// This function has been automatically generated from the project information.
{attribute 'signature_flag' := '1073741824'}
{attribute 'TcGenerated'}
{attribute 'no-analysis'}
FUNCTION F_GetTitle : WSTRING
VAR_INPUT
	
END_VAR

F_GetTitle := "Motion Library";

END_FUNCTION

(* stored: Version 1.1.0.1
   POU F_GetTitle: Id {c210cf97-aa66-408b-beb4-809f283b95e5}, SpecialFunc None *)
